(* IEC 61131-3 sources: hydraulic-pressure-control-codesys/src, 4 files *)

(* ---- GVL.st ---- *)
VAR_GLOBAL
    (* Pressure sensors — raw 4-20mA scaled to bar *)
    rPressure1      : REAL;   (* Inlet pressure *)
    rPressure2      : REAL;   (* Working pressure *)
    rPressure3      : REAL;   (* Return line pressure *)

    (* Proportional valve output 0.0-100.0% *)
    rValveOutput    : REAL;

    (* System state *)
    bSystemRun      : BOOL;
    bEmergencyStop  : BOOL;
    bFault          : BOOL;
    sFaultCode      : STRING;
END_VAR

(* ---- FB_HydraulicControl.st ---- *)
FUNCTION_BLOCK FB_HydraulicControl
VAR_INPUT
    bRun            : BOOL;
    bEStop          : BOOL;
    rPressure1      : REAL;
    rPressure2      : REAL;
    rPressure3      : REAL;
    rSetpoint       : REAL;         (* Target working pressure, bar *)
    rMaxPressure    : REAL := 200.0;
END_VAR
VAR_OUTPUT
    rValveOut       : REAL;         (* 0.0-100.0% *)
    bFault          : BOOL;
    sFaultCode      : STRING;
END_VAR
VAR
    PID             : FB_PID;
    bPIDEnable      : BOOL;
END_VAR

(* Emergency stop or active fault — close valve immediately *)
IF bEStop OR bFault THEN
    rValveOut  := 0.0;
    bPIDEnable := FALSE;
    RETURN;
END_IF

(* Overpressure protection *)
IF rPressure2 > rMaxPressure THEN
    bFault     := TRUE;
    sFaultCode := 'ERR_OVERPRESSURE_P2';
    rValveOut  := 0.0;
    RETURN;
END_IF

(* Wire break on any sensor *)
IF rPressure1 <= 0.0 OR rPressure2 <= 0.0 OR rPressure3 <= 0.0 THEN
    bFault     := TRUE;
    sFaultCode := 'ERR_SENSOR_FAULT';
    rValveOut  := 0.0;
    RETURN;
END_IF

(* Normal run — PID controls proportional valve *)
bPIDEnable := bRun;
PID(
    bEnable        := bPIDEnable,
    fSetpointValue := rSetpoint,
    fActualValue   := rPressure2,
    fManSyncValue  := 0.0,
    eMode          := ePID_Mode.Active,
    fOut           => rValveOut
);

rValveOut := LIMIT(0.0, rValveOut, 100.0);

(* ---- FB_PressureScale.st ---- *)
FUNCTION_BLOCK FB_PressureScale
VAR_INPUT
    iRawADC     : INT;      (* 0-32767 from AI module *)
    rMinBar     : REAL;     (* Engineering min, e.g. 0.0 *)
    rMaxBar     : REAL;     (* Engineering max, e.g. 250.0 *)
END_VAR
VAR_OUTPUT
    rPressure   : REAL;
    bWireBroken : BOOL;     (* TRUE if signal < 3.8 mA *)
END_VAR
VAR
    rScaled     : REAL;
END_VAR

(* 4mA = ~6554, 20mA = 32767 on 0-32767 range *)
IF iRawADC < 5900 THEN
    bWireBroken := TRUE;
    rPressure   := 0.0;
ELSE
    bWireBroken := FALSE;
    rScaled := (INT_TO_REAL(iRawADC) - 6554.0) / (32767.0 - 6554.0);
    rPressure := rMinBar + rScaled * (rMaxBar - rMinBar);
    rPressure := LIMIT(rMinBar, rPressure, rMaxBar);
END_IF

(* ---- MAIN.st ---- *)
PROGRAM MAIN
VAR
    Scale1    : FB_PressureScale;
    Scale2    : FB_PressureScale;
    Scale3    : FB_PressureScale;
    Hydraulic : FB_HydraulicControl;

    (* Simulated ADC inputs — connect to real AI channels in production *)
    iADC1     : INT := 16000;
    iADC2     : INT := 18000;
    iADC3     : INT := 14000;
END_VAR

(* Scale 4-20mA sensor signals to bar *)
Scale1(iRawADC := iADC1, rMinBar := 0.0, rMaxBar := 250.0, rPressure => GVL.rPressure1);
Scale2(iRawADC := iADC2, rMinBar := 0.0, rMaxBar := 250.0, rPressure => GVL.rPressure2);
Scale3(iRawADC := iADC3, rMinBar := 0.0, rMaxBar := 250.0, rPressure => GVL.rPressure3);

(* Hydraulic control with PID and fault handling *)
Hydraulic(
    bRun       := GVL.bSystemRun,
    bEStop     := GVL.bEmergencyStop,
    rPressure1 := GVL.rPressure1,
    rPressure2 := GVL.rPressure2,
    rPressure3 := GVL.rPressure3,
    rSetpoint  := 120.0,
    rValveOut  => GVL.rValveOutput,
    bFault     => GVL.bFault,
    sFaultCode => GVL.sFaultCode
);
